Fanuc KAREL source: kt00298.KL

PROGRAM KT00298
%NOLOCKGROUP
VAR
R1:REAL;R2:REAL;OUT:BOOLEAN
BEGIN
--
--
R1=2.0
R2=3.0
R1=2.0
R2=3.0
OUT=(R1<>R2)
END KT00298
